FUNCTION_BLOCK RampUp
VAR_INPUT
    Setpoint    : REAL;    // Target value to ramp up to
    RampUpTime  : TIME;    // Time to ramp up to the setpoint
    Enable      : BOOL;    // Enables the ramping process
END_VAR

VAR_OUTPUT
    Output      : REAL;    // Current output value
    InProgress  : BOOL;    // TRUE while ramping is in progress
END_VAR

VAR
    StartValue  : REAL;    // Starting value of the ramp
    RampRate    : REAL;    // Rate of change per second
    ElapsedTime : TIME;    // Time passed since the start of the ramp
    Timer       : TON;     // Timer for tracking elapsed time
END_VAR


// Initialize ramp if enabled
IF Enable THEN
    IF NOT InProgress THEN
        // Start ramping
        StartValue := Output;
        Timer(IN := TRUE, PT := RampUpTime); // Start the timer
        
        IF RampUpTime > T#0S THEN
            // Calculate ramp rate
            RampRate := (Setpoint - StartValue) / TIME_TO_REAL(RampUpTime);
        ELSE
            RampRate := Setpoint - StartValue;
        END_IF
        
        InProgress := TRUE;
    END_IF

    // Update elapsed time from the timer
    ElapsedTime := Timer.ET; // ET is the elapsed time of the timer
    
    // Check if the ramp time has been reached
    IF Timer.Q THEN
        Output := Setpoint;  // Set the output to the target value
        InProgress := FALSE; // Ramp process is complete
    ELSE
        // Incrementally update the output
        Output := StartValue + TIME_TO_REAL(ElapsedTime) * RampRate;
    END_IF
ELSE
    InProgress := FALSE;
    Timer(IN := FALSE); // Stop the timer if ramping is disabled
	Output	:=	0;
END_IF

Timer();

END_FUNCTION_BLOCK

(* stored: Version 1.1.0.1, ProductVersion 3.1.4024.13
   POU RampUp: Id {f2658a87-6266-4377-b780-07aa5b994daa}, SpecialFunc None *)
